// TwinCAT 3 PLC project PLC
// ProgramVersion: 3.1.4024.0
// libraries:
//   EfficientIO Communicator, * (EfficientIO)
//   Lynus Energy Basic, * (Lynus AG)
//   Lynus Persistent Data V1, * (Lynus AG)
//   Lynus Standards, * (Lynus AG)
//   Tc2_Standard, * (Beckhoff Automation GmbH)
//   Tc2_System, * (Beckhoff Automation GmbH)
//   Tc3_IPCDiag, * (Beckhoff Automation GmbH)
//   Tc3_Module, * (Beckhoff Automation GmbH)
// project tree:
//   ENUMs/ E_State.TcDUT (not stored)
//   / FastTask.TcTTO, MiddleTask.TcTTO, SlowTask.TcTTO (not stored)
//   POUs/ prgComEffIO.TcPOU, prgEM.TcPOU, prgOutputs.TcPOU, prgRWEffIO.TcPOU (not stored), prgVarEffIO.TcPOU (not stored), prg_ReadDeviceName.TcPOU (not stored)
// real-time tasks:
//   TASK PlcTask: cycle T#10ms, priority 20, ADS port 350
//   TASK FastTask: cycle T#5ms, priority 19, ADS port 351
//   TASK MiddleTask: cycle T#10ms, priority 21, ADS port 352
//   TASK SlowTask: cycle T#20ms, priority 23, ADS port 353
// I/O:
//   DEVICE Gerät 2 (CX-BK)
//     Box 1 (CX-BK)
// variable links:
//   PLC/PLC Instance <-> Device 2 (CX-BK)/Box 1 (CX-BK)
//     MiddleTask Inputs/prgEM.fbEM1.fbKL3403.byStateCH1 <-> Term 2 (KL3403)/Channel 1/Status
//     MiddleTask Inputs/prgEM.fbEM1.fbKL3403.byStateCH2 <-> Term 2 (KL3403)/Channel 2/Status
//     MiddleTask Inputs/prgEM.fbEM1.fbKL3403.byStateCH3 <-> Term 2 (KL3403)/Channel 3/Status
//     MiddleTask Inputs/prgEM.fbEM10.fbKL3403.byStateCH1 <-> Term 11 (KL3403)/Channel 1/Status
//     MiddleTask Inputs/prgEM.fbEM10.fbKL3403.byStateCH2 <-> Term 11 (KL3403)/Channel 2/Status
//     MiddleTask Inputs/prgEM.fbEM10.fbKL3403.byStateCH3 <-> Term 11 (KL3403)/Channel 3/Status
//     MiddleTask Inputs/prgEM.fbEM11.fbKL3403.byStateCH1 <-> Term 12 (KL3403)/Channel 1/Status
//     MiddleTask Inputs/prgEM.fbEM11.fbKL3403.byStateCH2 <-> Term 12 (KL3403)/Channel 2/Status
//     MiddleTask Inputs/prgEM.fbEM11.fbKL3403.byStateCH3 <-> Term 12 (KL3403)/Channel 3/Status
//     MiddleTask Inputs/prgEM.fbEM12.fbKL3403.byStateCH1 <-> Term 13 (KL3403)/Channel 1/Status
//     MiddleTask Inputs/prgEM.fbEM12.fbKL3403.byStateCH2 <-> Term 13 (KL3403)/Channel 2/Status
//     MiddleTask Inputs/prgEM.fbEM12.fbKL3403.byStateCH3 <-> Term 13 (KL3403)/Channel 3/Status
//     MiddleTask Inputs/prgEM.fbEM2.fbKL3403.byStateCH1 <-> Term 3 (KL3403)/Channel 1/Status
//     MiddleTask Inputs/prgEM.fbEM2.fbKL3403.byStateCH2 <-> Term 3 (KL3403)/Channel 2/Status
//     MiddleTask Inputs/prgEM.fbEM2.fbKL3403.byStateCH3 <-> Term 3 (KL3403)/Channel 3/Status
//     MiddleTask Inputs/prgEM.fbEM3.fbKL3403.byStateCH1 <-> Term 4 (KL3403)/Channel 1/Status
//     MiddleTask Inputs/prgEM.fbEM3.fbKL3403.byStateCH2 <-> Term 4 (KL3403)/Channel 2/Status
//     MiddleTask Inputs/prgEM.fbEM3.fbKL3403.byStateCH3 <-> Term 4 (KL3403)/Channel 3/Status
//     MiddleTask Inputs/prgEM.fbEM4.fbKL3403.byStateCH1 <-> Term 5 (KL3403)/Channel 1/Status
//     MiddleTask Inputs/prgEM.fbEM4.fbKL3403.byStateCH2 <-> Term 5 (KL3403)/Channel 2/Status
//     MiddleTask Inputs/prgEM.fbEM4.fbKL3403.byStateCH3 <-> Term 5 (KL3403)/Channel 3/Status
//     MiddleTask Inputs/prgEM.fbEM5.fbKL3403.byStateCH1 <-> Term 6 (KL3403)/Channel 1/Status
//     MiddleTask Inputs/prgEM.fbEM5.fbKL3403.byStateCH2 <-> Term 6 (KL3403)/Channel 2/Status
//     MiddleTask Inputs/prgEM.fbEM5.fbKL3403.byStateCH3 <-> Term 6 (KL3403)/Channel 3/Status
//     MiddleTask Inputs/prgEM.fbEM6.fbKL3403.byStateCH1 <-> Term 7 (KL3403)/Channel 1/Status
//     MiddleTask Inputs/prgEM.fbEM6.fbKL3403.byStateCH2 <-> Term 7 (KL3403)/Channel 2/Status
//     MiddleTask Inputs/prgEM.fbEM6.fbKL3403.byStateCH3 <-> Term 7 (KL3403)/Channel 3/Status
//     MiddleTask Inputs/prgEM.fbEM7.fbKL3403.byStateCH1 <-> Term 8 (KL3403)/Channel 1/Status
//     MiddleTask Inputs/prgEM.fbEM7.fbKL3403.byStateCH2 <-> Term 8 (KL3403)/Channel 2/Status
//     MiddleTask Inputs/prgEM.fbEM7.fbKL3403.byStateCH3 <-> Term 8 (KL3403)/Channel 3/Status
//     MiddleTask Inputs/prgEM.fbEM8.fbKL3403.byStateCH1 <-> Term 9 (KL3403)/Channel 1/Status
//     MiddleTask Inputs/prgEM.fbEM8.fbKL3403.byStateCH2 <-> Term 9 (KL3403)/Channel 2/Status
//     MiddleTask Inputs/prgEM.fbEM8.fbKL3403.byStateCH3 <-> Term 9 (KL3403)/Channel 3/Status
//     MiddleTask Inputs/prgEM.fbEM9.fbKL3403.byStateCH1 <-> Term 10 (KL3403)/Channel 1/Status
//     MiddleTask Inputs/prgEM.fbEM9.fbKL3403.byStateCH2 <-> Term 10 (KL3403)/Channel 2/Status
//     MiddleTask Inputs/prgEM.fbEM9.fbKL3403.byStateCH3 <-> Term 10 (KL3403)/Channel 3/Status
//     MiddleTask Inputs/prgEM.fbEM1.fbKL3403.iDataInCH1 <-> Term 2 (KL3403)/Channel 1/Daten Ein
//     MiddleTask Inputs/prgEM.fbEM1.fbKL3403.iDataInCH2 <-> Term 2 (KL3403)/Channel 2/Daten Ein
//     MiddleTask Inputs/prgEM.fbEM1.fbKL3403.iDataInCH3 <-> Term 2 (KL3403)/Channel 3/Daten Ein
//     MiddleTask Inputs/prgEM.fbEM10.fbKL3403.iDataInCH1 <-> Term 11 (KL3403)/Channel 1/Daten Ein
//     MiddleTask Inputs/prgEM.fbEM10.fbKL3403.iDataInCH2 <-> Term 11 (KL3403)/Channel 2/Daten Ein
//     MiddleTask Inputs/prgEM.fbEM10.fbKL3403.iDataInCH3 <-> Term 11 (KL3403)/Channel 3/Daten Ein
//     MiddleTask Inputs/prgEM.fbEM11.fbKL3403.iDataInCH1 <-> Term 12 (KL3403)/Channel 1/Daten Ein
//     MiddleTask Inputs/prgEM.fbEM11.fbKL3403.iDataInCH2 <-> Term 12 (KL3403)/Channel 2/Daten Ein
//     MiddleTask Inputs/prgEM.fbEM11.fbKL3403.iDataInCH3 <-> Term 12 (KL3403)/Channel 3/Daten Ein
//     MiddleTask Inputs/prgEM.fbEM12.fbKL3403.iDataInCH1 <-> Term 13 (KL3403)/Channel 1/Daten Ein
//     MiddleTask Inputs/prgEM.fbEM12.fbKL3403.iDataInCH2 <-> Term 13 (KL3403)/Channel 2/Daten Ein
//     MiddleTask Inputs/prgEM.fbEM12.fbKL3403.iDataInCH3 <-> Term 13 (KL3403)/Channel 3/Daten Ein
//     MiddleTask Inputs/prgEM.fbEM2.fbKL3403.iDataInCH1 <-> Term 3 (KL3403)/Channel 1/Daten Ein
//     MiddleTask Inputs/prgEM.fbEM2.fbKL3403.iDataInCH2 <-> Term 3 (KL3403)/Channel 2/Daten Ein
//     MiddleTask Inputs/prgEM.fbEM2.fbKL3403.iDataInCH3 <-> Term 3 (KL3403)/Channel 3/Daten Ein
//     MiddleTask Inputs/prgEM.fbEM3.fbKL3403.iDataInCH1 <-> Term 4 (KL3403)/Channel 1/Daten Ein
//     MiddleTask Inputs/prgEM.fbEM3.fbKL3403.iDataInCH2 <-> Term 4 (KL3403)/Channel 2/Daten Ein
//     MiddleTask Inputs/prgEM.fbEM3.fbKL3403.iDataInCH3 <-> Term 4 (KL3403)/Channel 3/Daten Ein
//     MiddleTask Inputs/prgEM.fbEM4.fbKL3403.iDataInCH1 <-> Term 5 (KL3403)/Channel 1/Daten Ein
//     MiddleTask Inputs/prgEM.fbEM4.fbKL3403.iDataInCH2 <-> Term 5 (KL3403)/Channel 2/Daten Ein
//     MiddleTask Inputs/prgEM.fbEM4.fbKL3403.iDataInCH3 <-> Term 5 (KL3403)/Channel 3/Daten Ein
//     MiddleTask Inputs/prgEM.fbEM5.fbKL3403.iDataInCH1 <-> Term 6 (KL3403)/Channel 1/Daten Ein
//     MiddleTask Inputs/prgEM.fbEM5.fbKL3403.iDataInCH2 <-> Term 6 (KL3403)/Channel 2/Daten Ein
//     MiddleTask Inputs/prgEM.fbEM5.fbKL3403.iDataInCH3 <-> Term 6 (KL3403)/Channel 3/Daten Ein
//     MiddleTask Inputs/prgEM.fbEM6.fbKL3403.iDataInCH1 <-> Term 7 (KL3403)/Channel 1/Daten Ein
//     MiddleTask Inputs/prgEM.fbEM6.fbKL3403.iDataInCH2 <-> Term 7 (KL3403)/Channel 2/Daten Ein
//     MiddleTask Inputs/prgEM.fbEM6.fbKL3403.iDataInCH3 <-> Term 7 (KL3403)/Channel 3/Daten Ein
//     MiddleTask Inputs/prgEM.fbEM7.fbKL3403.iDataInCH1 <-> Term 8 (KL3403)/Channel 1/Daten Ein
//     MiddleTask Inputs/prgEM.fbEM7.fbKL3403.iDataInCH2 <-> Term 8 (KL3403)/Channel 2/Daten Ein
//     MiddleTask Inputs/prgEM.fbEM7.fbKL3403.iDataInCH3 <-> Term 8 (KL3403)/Channel 3/Daten Ein
//     MiddleTask Inputs/prgEM.fbEM8.fbKL3403.iDataInCH1 <-> Term 9 (KL3403)/Channel 1/Daten Ein
//     MiddleTask Inputs/prgEM.fbEM8.fbKL3403.iDataInCH2 <-> Term 9 (KL3403)/Channel 2/Daten Ein
//     MiddleTask Inputs/prgEM.fbEM8.fbKL3403.iDataInCH3 <-> Term 9 (KL3403)/Channel 3/Daten Ein
//     MiddleTask Inputs/prgEM.fbEM9.fbKL3403.iDataInCH1 <-> Term 10 (KL3403)/Channel 1/Daten Ein
//     MiddleTask Inputs/prgEM.fbEM9.fbKL3403.iDataInCH2 <-> Term 10 (KL3403)/Channel 2/Daten Ein
//     MiddleTask Inputs/prgEM.fbEM9.fbKL3403.iDataInCH3 <-> Term 10 (KL3403)/Channel 3/Daten Ein
//     MiddleTask Inputs/prgEM.fbKBusState.uiKBusState_OUT <-> Inputs/State
//     MiddleTask Outputs/prgEM.fbEM1.fbKL3403.byCntrCH1 <-> Term 2 (KL3403)/Channel 1/Kontrolle
//     MiddleTask Outputs/prgEM.fbEM1.fbKL3403.byCntrCH2 <-> Term 2 (KL3403)/Channel 2/Kontrolle
//     MiddleTask Outputs/prgEM.fbEM1.fbKL3403.byCntrCH3 <-> Term 2 (KL3403)/Channel 3/Kontrolle
//     MiddleTask Outputs/prgEM.fbEM10.fbKL3403.byCntrCH1 <-> Term 11 (KL3403)/Channel 1/Kontrolle
//     MiddleTask Outputs/prgEM.fbEM10.fbKL3403.byCntrCH2 <-> Term 11 (KL3403)/Channel 2/Kontrolle
//     MiddleTask Outputs/prgEM.fbEM10.fbKL3403.byCntrCH3 <-> Term 11 (KL3403)/Channel 3/Kontrolle
//     MiddleTask Outputs/prgEM.fbEM11.fbKL3403.byCntrCH1 <-> Term 12 (KL3403)/Channel 1/Kontrolle
//     MiddleTask Outputs/prgEM.fbEM11.fbKL3403.byCntrCH2 <-> Term 12 (KL3403)/Channel 2/Kontrolle
//     MiddleTask Outputs/prgEM.fbEM11.fbKL3403.byCntrCH3 <-> Term 12 (KL3403)/Channel 3/Kontrolle
//     MiddleTask Outputs/prgEM.fbEM12.fbKL3403.byCntrCH1 <-> Term 13 (KL3403)/Channel 1/Kontrolle
//     MiddleTask Outputs/prgEM.fbEM12.fbKL3403.byCntrCH2 <-> Term 13 (KL3403)/Channel 2/Kontrolle
//     MiddleTask Outputs/prgEM.fbEM12.fbKL3403.byCntrCH3 <-> Term 13 (KL3403)/Channel 3/Kontrolle
//     MiddleTask Outputs/prgEM.fbEM2.fbKL3403.byCntrCH1 <-> Term 3 (KL3403)/Channel 1/Kontrolle
//     MiddleTask Outputs/prgEM.fbEM2.fbKL3403.byCntrCH2 <-> Term 3 (KL3403)/Channel 2/Kontrolle
//     MiddleTask Outputs/prgEM.fbEM2.fbKL3403.byCntrCH3 <-> Term 3 (KL3403)/Channel 3/Kontrolle
//     MiddleTask Outputs/prgEM.fbEM3.fbKL3403.byCntrCH1 <-> Term 4 (KL3403)/Channel 1/Kontrolle
//     MiddleTask Outputs/prgEM.fbEM3.fbKL3403.byCntrCH2 <-> Term 4 (KL3403)/Channel 2/Kontrolle
//     MiddleTask Outputs/prgEM.fbEM3.fbKL3403.byCntrCH3 <-> Term 4 (KL3403)/Channel 3/Kontrolle
//     MiddleTask Outputs/prgEM.fbEM4.fbKL3403.byCntrCH1 <-> Term 5 (KL3403)/Channel 1/Kontrolle
//     MiddleTask Outputs/prgEM.fbEM4.fbKL3403.byCntrCH2 <-> Term 5 (KL3403)/Channel 2/Kontrolle
//     MiddleTask Outputs/prgEM.fbEM4.fbKL3403.byCntrCH3 <-> Term 5 (KL3403)/Channel 3/Kontrolle
//     MiddleTask Outputs/prgEM.fbEM5.fbKL3403.byCntrCH1 <-> Term 6 (KL3403)/Channel 1/Kontrolle
//     MiddleTask Outputs/prgEM.fbEM5.fbKL3403.byCntrCH2 <-> Term 6 (KL3403)/Channel 2/Kontrolle
//     MiddleTask Outputs/prgEM.fbEM5.fbKL3403.byCntrCH3 <-> Term 6 (KL3403)/Channel 3/Kontrolle
//     MiddleTask Outputs/prgEM.fbEM6.fbKL3403.byCntrCH1 <-> Term 7 (KL3403)/Channel 1/Kontrolle
//     MiddleTask Outputs/prgEM.fbEM6.fbKL3403.byCntrCH2 <-> Term 7 (KL3403)/Channel 2/Kontrolle
//     MiddleTask Outputs/prgEM.fbEM6.fbKL3403.byCntrCH3 <-> Term 7 (KL3403)/Channel 3/Kontrolle
//     MiddleTask Outputs/prgEM.fbEM7.fbKL3403.byCntrCH1 <-> Term 8 (KL3403)/Channel 1/Kontrolle
//     MiddleTask Outputs/prgEM.fbEM7.fbKL3403.byCntrCH2 <-> Term 8 (KL3403)/Channel 2/Kontrolle
//     MiddleTask Outputs/prgEM.fbEM7.fbKL3403.byCntrCH3 <-> Term 8 (KL3403)/Channel 3/Kontrolle
//     MiddleTask Outputs/prgEM.fbEM8.fbKL3403.byCntrCH1 <-> Term 9 (KL3403)/Channel 1/Kontrolle
//     MiddleTask Outputs/prgEM.fbEM8.fbKL3403.byCntrCH2 <-> Term 9 (KL3403)/Channel 2/Kontrolle
//     MiddleTask Outputs/prgEM.fbEM8.fbKL3403.byCntrCH3 <-> Term 9 (KL3403)/Channel 3/Kontrolle
//     MiddleTask Outputs/prgEM.fbEM9.fbKL3403.byCntrCH1 <-> Term 10 (KL3403)/Channel 1/Kontrolle
//     MiddleTask Outputs/prgEM.fbEM9.fbKL3403.byCntrCH2 <-> Term 10 (KL3403)/Channel 2/Kontrolle
//     MiddleTask Outputs/prgEM.fbEM9.fbKL3403.byCntrCH3 <-> Term 10 (KL3403)/Channel 3/Kontrolle
//     MiddleTask Outputs/prgOutputs.mOut_1_1 <-> Term 14 (KL2012)/Channel 1/Ausgang
//     MiddleTask Outputs/prgOutputs.mOut_1_2 <-> Term 14 (KL2012)/Channel 2/Ausgang
//     MiddleTask Outputs/prgOutputs.mOut_2_1 <-> Term 15 (KL2012)/Channel 1/Ausgang
//     MiddleTask Outputs/prgOutputs.mOut_2_2 <-> Term 15 (KL2012)/Channel 2/Ausgang
//     MiddleTask Outputs/prgOutputs.mOut_3_1 <-> Term 16 (KL2012)/Channel 1/Ausgang
//     MiddleTask Outputs/prgOutputs.mOut_3_2 <-> Term 16 (KL2012)/Channel 2/Ausgang
//     MiddleTask Outputs/prgOutputs.mOut_4_1 <-> Term 17 (KL2012)/Channel 1/Ausgang
//     MiddleTask Outputs/prgOutputs.mOut_4_2 <-> Term 17 (KL2012)/Channel 2/Ausgang

CONFIGURATION PLC
    RESOURCE PLC ON TwinCAT3
        TASK FastTask(INTERVAL := T#5ms, PRIORITY := 19);
        TASK MiddleTask(INTERVAL := T#10ms, PRIORITY := 21);
        PROGRAM prgRWEffIO WITH FastTask : prgRWEffIO;
        PROGRAM prgVarEffIO WITH FastTask : prgVarEffIO;
        PROGRAM prgEM WITH MiddleTask : prgEM;
        PROGRAM prgOutputs WITH MiddleTask : prgOutputs;
    END_RESOURCE
END_CONFIGURATION

// ---- POUs/prgEM.TcPOU
PROGRAM prgEM
VAR
	fbKBusState		: FB_K_Bus_State;
	fbEM1			: FB_EM_Beckhoff_KL3403;
	fbEM1Counter	: FB_EnergyCounter;
	fbEM2			: FB_EM_Beckhoff_KL3403;
	fbEM2Counter	: FB_EnergyCounter;
	fbEM3			: FB_EM_Beckhoff_KL3403;
	fbEM3Counter	: FB_EnergyCounter;
	fbEM4			: FB_EM_Beckhoff_KL3403;
	fbEM4Counter	: FB_EnergyCounter;
	fbEM5			: FB_EM_Beckhoff_KL3403;
	fbEM5Counter	: FB_EnergyCounter;
	fbEM6			: FB_EM_Beckhoff_KL3403;
	fbEM6Counter	: FB_EnergyCounter;
	fbEM7			: FB_EM_Beckhoff_KL3403;
	fbEM7Counter	: FB_EnergyCounter;
	fbEM8			: FB_EM_Beckhoff_KL3403;
	fbEM8Counter	: FB_EnergyCounter;
	fbEM9			: FB_EM_Beckhoff_KL3403;
	fbEM9Counter	: FB_EnergyCounter;
	fbEM10			: FB_EM_Beckhoff_KL3403;
	fbEM10Counter	: FB_EnergyCounter;
	fbEM11			: FB_EM_Beckhoff_KL3403;
	fbEM11Counter	: FB_EnergyCounter;
	fbEM12			: FB_EM_Beckhoff_KL3403;
	fbEM12Counter	: FB_EnergyCounter;
	
	lrPowerEM1		: LREAL;						//{#lynus.ag#()}
	lrPowerEM2		: LREAL;						//{#lynus.ag#()}
	lrPowerEM3		: LREAL;						//{#lynus.ag#()}
	lrPowerEM4		: LREAL;						//{#lynus.ag#()}
	lrPowerEM5		: LREAL;						//{#lynus.ag#()}
	lrPowerEM6		: LREAL;						//{#lynus.ag#()}
	lrPowerEM7		: LREAL;						//{#lynus.ag#()}
	lrPowerEM8		: LREAL;						//{#lynus.ag#()}
	lrPowerEM9		: LREAL;						//{#lynus.ag#()}
	lrPowerEM10		: LREAL;						//{#lynus.ag#()}
	lrPowerEM11		: LREAL;						//{#lynus.ag#()}
	lrPowerEM12		: LREAL;						//{#lynus.ag#()}
	lr_InputVoltage_L1N		: LREAL;						//{#lynus.ag#()}
	lr_InputVoltage_L2N		: LREAL;						//{#lynus.ag#()}
	lr_InputVoltage_L3N		: LREAL;						//{#lynus.ag#()}
	lr_InputVoltage_L1L2	: LREAL;						//{#lynus.ag#()}
	lr_InputVoltage_L2L3	: LREAL;						//{#lynus.ag#()}
	lr_InputVoltage_L3L1	: LREAL;						//{#lynus.ag#()}
	lr_FrequencyEM1			: LREAL;						//{#lynus.ag#()}
	lr_CurrentL1EM1			: LREAL;						//{#lynus.ag#()}
	lr_CurrentL2EM1			: LREAL;						//{#lynus.ag#()}
	lr_CurrentL3EM1			: LREAL;						//{#lynus.ag#()}
END_VAR
VAR_INPUT
	uiCurrentTransformerRatio_EM1	:UINT:=400;			// unklar ob korrekt
	uiCurrentTransformerRatio_EM2	:UINT:=400;			// unklar ob korrekt
	uiCurrentTransformerRatio_EM3	:UINT:=250;
	uiCurrentTransformerRatio_EM4	:UINT:=64;
	uiCurrentTransformerRatio_EM5	:UINT:=64;
	uiCurrentTransformerRatio_EM6	:UINT:=35;
	uiCurrentTransformerRatio_EM7	:UINT:=35;
	uiCurrentTransformerRatio_EM8	:UINT:=35;
	uiCurrentTransformerRatio_EM9	:UINT:=35;
	uiCurrentTransformerRatio_EM10	:UINT:=35;
	uiCurrentTransformerRatio_EM11	:UINT:=35;
	uiCurrentTransformerRatio_EM12	:UINT:=35;

END_VAR
VAR PERSISTENT
	lrCounterEM1	: LREAL;						//{#lynus.ag#()}
	lrCounterEM2	: LREAL;						//{#lynus.ag#()}
	lrCounterEM3	: LREAL;						//{#lynus.ag#()}
	lrCounterEM4	: LREAL;						//{#lynus.ag#()}
	lrCounterEM5	: LREAL;						//{#lynus.ag#()}
	lrCounterEM6	: LREAL;						//{#lynus.ag#()}
	lrCounterEM7	: LREAL;						//{#lynus.ag#()}
	lrCounterEM8	: LREAL;						//{#lynus.ag#()}
	lrCounterEM9	: LREAL;						//{#lynus.ag#()}
	lrCounterEM10	: LREAL;						//{#lynus.ag#()}
	lrCounterEM11	: LREAL;						//{#lynus.ag#()}
	lrCounterEM12	: LREAL;						//{#lynus.ag#()}
END_VAR

fbKBusState(	uiKBusState_OUT=> , 
				b_Kbus_notOk=> , 
				word_ErrorCount=> );


fbEM1(
	bEnable:= TRUE, 
	bChannel1Invers:= FALSE,
	bChannel2Invers:= FALSE,
	bChannel3Invers:= FALSE,
	uiCurrentTransformerRatioL1:= uiCurrentTransformerRatio_EM1, 
	uiCurrentTransformerRatioL2:= uiCurrentTransformerRatio_EM1, 
	uiCurrentTransformerRatioL3:= uiCurrentTransformerRatio_EM1, 
	uiKBusState_IN:= fbKBusState.uiKBusState_OUT, 
	stDataEMPower=> , 
	stDataEMCounter=> , 
	stDataEMPowerRealTime=> , 
	stDataEMCounterRealTime=> , 
	diNrOfEM_OUT=> );

lrPowerEM1 := fbEM1.stDataEMPower.lrPowerTotal;	
lr_InputVoltage_L1N := fbEM1.stDataEMPower.lrVoltageL1N;
lr_InputVoltage_L2N := fbEM1.stDataEMPower.lrVoltageL2N;
lr_InputVoltage_L3N := fbEM1.stDataEMPower.lrVoltageL3N;
lr_InputVoltage_L1L2 := fbEM1.stDataEMPower.lrVoltageL1L2;
lr_InputVoltage_L2L3 := fbEM1.stDataEMPower.lrVoltageL2L3;
lr_InputVoltage_L3L1 := fbEM1.stDataEMPower.lrVoltageL3L1;
lr_FrequencyEM1		:= fbEM1.stDataEMPower.lrFrequency;
lr_CurrentL1EM1		:= fbEM1.stDataEMPower.lrCurrentL1;
lr_CurrentL2EM1		:= fbEM1.stDataEMPower.lrCurrentL2;
lr_CurrentL3EM1		:= fbEM1.stDataEMPower.lrCurrentL3;

fbEM1Counter(
	byActiveTariff:= 1, 
	lrPowerInput:= lrPowerEM1, 
	lrTotalCounterEnergy_Consumption=> , 
	lrTotalCounterEnergy_Production=> , 
	lrCounterEnergyT1_Consumption=> , 
	lrCounterEnergyT2_Consumption=> , 
	lrCounterEnergyT1_Production=> , 
	lrCounterEnergyT2_Production=> );
	
IF fbEM1Counter.lrTotalCounterEnergy_Consumption > lrCounterEM1 THEN  	
	lrCounterEM1 := fbEM1Counter.lrTotalCounterEnergy_Consumption;
END_IF


fbEM2(
	bEnable:= TRUE, 
	bChannel1Invers:= FALSE,
	bChannel2Invers:= FALSE,
	bChannel3Invers:= FALSE,
	uiCurrentTransformerRatioL1:= uiCurrentTransformerRatio_EM2, 
	uiCurrentTransformerRatioL2:= uiCurrentTransformerRatio_EM2, 
	uiCurrentTransformerRatioL3:= uiCurrentTransformerRatio_EM2, 
	uiKBusState_IN:= fbKBusState.uiKBusState_OUT, 
	stDataEMPower=> , 
	stDataEMCounter=> , 
	stDataEMPowerRealTime=> , 
	stDataEMCounterRealTime=> , 
	diNrOfEM_OUT=> );

lrPowerEM2 := fbEM2.stDataEMPower.lrPowerTotal;	

fbEM2Counter(
	byActiveTariff:= 1, 
	lrPowerInput:= lrPowerEM2, 
	lrTotalCounterEnergy_Consumption=> , 
	lrTotalCounterEnergy_Production=> , 
	lrCounterEnergyT1_Consumption=> , 
	lrCounterEnergyT2_Consumption=> , 
	lrCounterEnergyT1_Production=> , 
	lrCounterEnergyT2_Production=> );
	
IF fbEM2Counter.lrTotalCounterEnergy_Consumption > lrCounterEM2 THEN  	
	lrCounterEM2 := fbEM2Counter.lrTotalCounterEnergy_Consumption;
END_IF


fbEM3(
	bEnable:= TRUE, 
	bChannel1Invers:= FALSE,
	bChannel2Invers:= FALSE,
	bChannel3Invers:= FALSE,
	uiCurrentTransformerRatioL1:= uiCurrentTransformerRatio_EM3, 
	uiCurrentTransformerRatioL2:= uiCurrentTransformerRatio_EM3, 
	uiCurrentTransformerRatioL3:= uiCurrentTransformerRatio_EM3, 
	uiKBusState_IN:= fbKBusState.uiKBusState_OUT, 
	stDataEMPower=> , 
	stDataEMCounter=> , 
	stDataEMPowerRealTime=> , 
	stDataEMCounterRealTime=> , 
	diNrOfEM_OUT=> );

lrPowerEM3 := fbEM3.stDataEMPower.lrPowerTotal;	

fbEM3Counter(
	byActiveTariff:= 1, 
	lrPowerInput:= lrPowerEM3, 
	lrTotalCounterEnergy_Consumption=> , 
	lrTotalCounterEnergy_Production=> , 
	lrCounterEnergyT1_Consumption=> , 
	lrCounterEnergyT2_Consumption=> , 
	lrCounterEnergyT1_Production=> , 
	lrCounterEnergyT2_Production=> );
	
IF fbEM3Counter.lrTotalCounterEnergy_Consumption > lrCounterEM3 THEN  	
	lrCounterEM3 := fbEM3Counter.lrTotalCounterEnergy_Consumption;
END_IF

fbEM4(
	bEnable:= TRUE, 
	bChannel1Invers:= FALSE,
	bChannel2Invers:= FALSE,
	bChannel3Invers:= FALSE,
	uiCurrentTransformerRatioL1:= uiCurrentTransformerRatio_EM4, 
	uiCurrentTransformerRatioL2:= uiCurrentTransformerRatio_EM4, 
	uiCurrentTransformerRatioL3:= uiCurrentTransformerRatio_EM4, 
	uiKBusState_IN:= fbKBusState.uiKBusState_OUT, 
	stDataEMPower=> , 
	stDataEMCounter=> , 
	stDataEMPowerRealTime=> , 
	stDataEMCounterRealTime=> , 
	diNrOfEM_OUT=> );

lrPowerEM4 := fbEM4.stDataEMPower.lrPowerTotal;	

fbEM4Counter(
	byActiveTariff:= 1, 
	lrPowerInput:= lrPowerEM4, 
	lrTotalCounterEnergy_Consumption=> , 
	lrTotalCounterEnergy_Production=> , 
	lrCounterEnergyT1_Consumption=> , 
	lrCounterEnergyT2_Consumption=> , 
	lrCounterEnergyT1_Production=> , 
	lrCounterEnergyT2_Production=> );
	
IF fbEM4Counter.lrTotalCounterEnergy_Consumption > lrCounterEM4 THEN  	
	lrCounterEM4 := fbEM4Counter.lrTotalCounterEnergy_Consumption;
END_IF

fbEM5(
	bEnable:= TRUE, 
	bChannel1Invers:= FALSE,
	bChannel2Invers:= FALSE,
	bChannel3Invers:= FALSE,
	uiCurrentTransformerRatioL1:= uiCurrentTransformerRatio_EM5, 
	uiCurrentTransformerRatioL2:= uiCurrentTransformerRatio_EM5, 
	uiCurrentTransformerRatioL3:= uiCurrentTransformerRatio_EM5, 
	uiKBusState_IN:= fbKBusState.uiKBusState_OUT, 
	stDataEMPower=> , 
	stDataEMCounter=> , 
	stDataEMPowerRealTime=> , 
	stDataEMCounterRealTime=> , 
	diNrOfEM_OUT=> );

lrPowerEM5 := fbEM5.stDataEMPower.lrPowerTotal;	

fbEM5Counter(
	byActiveTariff:= 1, 
	lrPowerInput:= lrPowerEM5, 
	lrTotalCounterEnergy_Consumption=> , 
	lrTotalCounterEnergy_Production=> , 
	lrCounterEnergyT1_Consumption=> , 
	lrCounterEnergyT2_Consumption=> , 
	lrCounterEnergyT1_Production=> , 
	lrCounterEnergyT2_Production=> );
	
IF fbEM5Counter.lrTotalCounterEnergy_Consumption > lrCounterEM5 THEN  	
	lrCounterEM5 := fbEM5Counter.lrTotalCounterEnergy_Consumption;
END_IF

fbEM6(
	bEnable:= TRUE, 
	bChannel1Invers:= FALSE,
	bChannel2Invers:= FALSE,
	bChannel3Invers:= FALSE,
	uiCurrentTransformerRatioL1:= uiCurrentTransformerRatio_EM6, 
	uiCurrentTransformerRatioL2:= uiCurrentTransformerRatio_EM6, 
	uiCurrentTransformerRatioL3:= uiCurrentTransformerRatio_EM6, 
	uiKBusState_IN:= fbKBusState.uiKBusState_OUT, 
	stDataEMPower=> , 
	stDataEMCounter=> , 
	stDataEMPowerRealTime=> , 
	stDataEMCounterRealTime=> , 
	diNrOfEM_OUT=> );

lrPowerEM6 := fbEM6.stDataEMPower.lrPowerTotal;	

fbEM6Counter(
	byActiveTariff:= 1, 
	lrPowerInput:= lrPowerEM6, 
	lrTotalCounterEnergy_Consumption=> , 
	lrTotalCounterEnergy_Production=> , 
	lrCounterEnergyT1_Consumption=> , 
	lrCounterEnergyT2_Consumption=> , 
	lrCounterEnergyT1_Production=> , 
	lrCounterEnergyT2_Production=> );
	
IF fbEM6Counter.lrTotalCounterEnergy_Consumption > lrCounterEM6 THEN  	
	lrCounterEM6 := fbEM6Counter.lrTotalCounterEnergy_Consumption;
END_IF

fbEM7(
	bEnable:= TRUE, 
	bChannel1Invers:= FALSE,
	bChannel2Invers:= FALSE,
	bChannel3Invers:= FALSE,
	uiCurrentTransformerRatioL1:= uiCurrentTransformerRatio_EM7, 
	uiCurrentTransformerRatioL2:= uiCurrentTransformerRatio_EM7, 
	uiCurrentTransformerRatioL3:= uiCurrentTransformerRatio_EM7, 
	uiKBusState_IN:= fbKBusState.uiKBusState_OUT, 
	stDataEMPower=> , 
	stDataEMCounter=> , 
	stDataEMPowerRealTime=> , 
	stDataEMCounterRealTime=> , 
	diNrOfEM_OUT=> );

lrPowerEM7 := fbEM7.stDataEMPower.lrPowerTotal;	

fbEM7Counter(
	byActiveTariff:= 1, 
	lrPowerInput:= lrPowerEM7, 
	lrTotalCounterEnergy_Consumption=> , 
	lrTotalCounterEnergy_Production=> , 
	lrCounterEnergyT1_Consumption=> , 
	lrCounterEnergyT2_Consumption=> , 
	lrCounterEnergyT1_Production=> , 
	lrCounterEnergyT2_Production=> );
	
IF fbEM7Counter.lrTotalCounterEnergy_Consumption > lrCounterEM7 THEN  	
	lrCounterEM7 := fbEM7Counter.lrTotalCounterEnergy_Consumption;
END_IF

fbEM8(
	bEnable:= TRUE, 
	bChannel1Invers:= FALSE,
	bChannel2Invers:= FALSE,
	bChannel3Invers:= FALSE,
	uiCurrentTransformerRatioL1:= uiCurrentTransformerRatio_EM8, 
	uiCurrentTransformerRatioL2:= uiCurrentTransformerRatio_EM8, 
	uiCurrentTransformerRatioL3:= uiCurrentTransformerRatio_EM8, 
	uiKBusState_IN:= fbKBusState.uiKBusState_OUT, 
	stDataEMPower=> , 
	stDataEMCounter=> , 
	stDataEMPowerRealTime=> , 
	stDataEMCounterRealTime=> , 
	diNrOfEM_OUT=> );

lrPowerEM8 := fbEM8.stDataEMPower.lrPowerTotal;	

fbEM8Counter(
	byActiveTariff:= 1, 
	lrPowerInput:= lrPowerEM8, 
	lrTotalCounterEnergy_Consumption=> , 
	lrTotalCounterEnergy_Production=> , 
	lrCounterEnergyT1_Consumption=> , 
	lrCounterEnergyT2_Consumption=> , 
	lrCounterEnergyT1_Production=> , 
	lrCounterEnergyT2_Production=> );
	
IF fbEM8Counter.lrTotalCounterEnergy_Consumption > lrCounterEM8 THEN  	
	lrCounterEM8 := fbEM8Counter.lrTotalCounterEnergy_Consumption;
END_IF

fbEM9(
	bEnable:= TRUE, 
	bChannel1Invers:= FALSE,
	bChannel2Invers:= FALSE,
	bChannel3Invers:= FALSE,
	uiCurrentTransformerRatioL1:= uiCurrentTransformerRatio_EM9, 
	uiCurrentTransformerRatioL2:= uiCurrentTransformerRatio_EM9, 
	uiCurrentTransformerRatioL3:= uiCurrentTransformerRatio_EM9, 
	uiKBusState_IN:= fbKBusState.uiKBusState_OUT, 
	stDataEMPower=> , 
	stDataEMCounter=> , 
	stDataEMPowerRealTime=> , 
	stDataEMCounterRealTime=> , 
	diNrOfEM_OUT=> );

lrPowerEM9 := fbEM9.stDataEMPower.lrPowerTotal;	

fbEM9Counter(
	byActiveTariff:= 1, 
	lrPowerInput:= lrPowerEM9, 
	lrTotalCounterEnergy_Consumption=> , 
	lrTotalCounterEnergy_Production=> , 
	lrCounterEnergyT1_Consumption=> , 
	lrCounterEnergyT2_Consumption=> , 
	lrCounterEnergyT1_Production=> , 
	lrCounterEnergyT2_Production=> );
	
IF fbEM9Counter.lrTotalCounterEnergy_Consumption > lrCounterEM9 THEN  	
	lrCounterEM9 := fbEM9Counter.lrTotalCounterEnergy_Consumption;
END_IF

fbEM10(
	bEnable:= TRUE, 
	bChannel1Invers:= FALSE,
	bChannel2Invers:= FALSE,
	bChannel3Invers:= FALSE,
	uiCurrentTransformerRatioL1:= uiCurrentTransformerRatio_EM10, 
	uiCurrentTransformerRatioL2:= uiCurrentTransformerRatio_EM10, 
	uiCurrentTransformerRatioL3:= uiCurrentTransformerRatio_EM10, 
	uiKBusState_IN:= fbKBusState.uiKBusState_OUT, 
	stDataEMPower=> , 
	stDataEMCounter=> , 
	stDataEMPowerRealTime=> , 
	stDataEMCounterRealTime=> , 
	diNrOfEM_OUT=> );

lrPowerEM10 := fbEM10.stDataEMPower.lrPowerTotal;	

fbEM10Counter(
	byActiveTariff:= 1, 
	lrPowerInput:= lrPowerEM10, 
	lrTotalCounterEnergy_Consumption=> , 
	lrTotalCounterEnergy_Production=> , 
	lrCounterEnergyT1_Consumption=> , 
	lrCounterEnergyT2_Consumption=> , 
	lrCounterEnergyT1_Production=> , 
	lrCounterEnergyT2_Production=> );
	
IF fbEM10Counter.lrTotalCounterEnergy_Consumption > lrCounterEM10 THEN  	
	lrCounterEM10 := fbEM10Counter.lrTotalCounterEnergy_Consumption;
END_IF

fbEM11(
	bEnable:= TRUE, 
	bChannel1Invers:= FALSE,
	bChannel2Invers:= FALSE,
	bChannel3Invers:= FALSE,
	uiCurrentTransformerRatioL1:= uiCurrentTransformerRatio_EM11, 
	uiCurrentTransformerRatioL2:= uiCurrentTransformerRatio_EM11, 
	uiCurrentTransformerRatioL3:= uiCurrentTransformerRatio_EM11, 
	uiKBusState_IN:= fbKBusState.uiKBusState_OUT, 
	stDataEMPower=> , 
	stDataEMCounter=> , 
	stDataEMPowerRealTime=> , 
	stDataEMCounterRealTime=> , 
	diNrOfEM_OUT=> );

lrPowerEM11 := fbEM11.stDataEMPower.lrPowerTotal;	

fbEM11Counter(
	byActiveTariff:= 1, 
	lrPowerInput:= lrPowerEM11, 
	lrTotalCounterEnergy_Consumption=> , 
	lrTotalCounterEnergy_Production=> , 
	lrCounterEnergyT1_Consumption=> , 
	lrCounterEnergyT2_Consumption=> , 
	lrCounterEnergyT1_Production=> , 
	lrCounterEnergyT2_Production=> );
	
IF fbEM11Counter.lrTotalCounterEnergy_Consumption > lrCounterEM11 THEN  	
	lrCounterEM11 := fbEM11Counter.lrTotalCounterEnergy_Consumption;
END_IF

fbEM12(
	bEnable:= TRUE, 
	bChannel1Invers:= FALSE,
	bChannel2Invers:= FALSE,
	bChannel3Invers:= FALSE,
	uiCurrentTransformerRatioL1:= uiCurrentTransformerRatio_EM12, 
	uiCurrentTransformerRatioL2:= uiCurrentTransformerRatio_EM12, 
	uiCurrentTransformerRatioL3:= uiCurrentTransformerRatio_EM12, 
	uiKBusState_IN:= fbKBusState.uiKBusState_OUT, 
	stDataEMPower=> , 
	stDataEMCounter=> , 
	stDataEMPowerRealTime=> , 
	stDataEMCounterRealTime=> , 
	diNrOfEM_OUT=> );

lrPowerEM12 := fbEM12.stDataEMPower.lrPowerTotal;	

fbEM12Counter(
	byActiveTariff:= 1, 
	lrPowerInput:= lrPowerEM12, 
	lrTotalCounterEnergy_Consumption=> , 
	lrTotalCounterEnergy_Production=> , 
	lrCounterEnergyT1_Consumption=> , 
	lrCounterEnergyT2_Consumption=> , 
	lrCounterEnergyT1_Production=> , 
	lrCounterEnergyT2_Production=> );
	
IF fbEM12Counter.lrTotalCounterEnergy_Consumption > lrCounterEM12 THEN  	
	lrCounterEM12 := fbEM12Counter.lrTotalCounterEnergy_Consumption;
END_IF

END_PROGRAM

// ---- POUs/prgOutputs.TcPOU
PROGRAM prgOutputs
VAR
	mOut_1_1		AT%Q*: BOOL;								//{#lynus.ag#()}
	mOut_1_2		AT%Q*: BOOL;								//{#lynus.ag#()}
	mOut_2_1		AT%Q*: BOOL;								//{#lynus.ag#()}
	mOut_2_2		AT%Q*: BOOL;								//{#lynus.ag#()}
	mOut_3_1		AT%Q*: BOOL;								//{#lynus.ag#()}
	mOut_3_2		AT%Q*: BOOL;								//{#lynus.ag#()}
	mOut_4_1		AT%Q*: BOOL;								//{#lynus.ag#()}
	mOut_4_2		AT%Q*: BOOL;								//{#lynus.ag#()}
	mOut_Command_1_1		:BOOL;								//{#lynus.ag#()}
	mOut_Command_1_2		:BOOL;								//{#lynus.ag#()}
	mOut_Command_2_1		:BOOL;								//{#lynus.ag#()}
	mOut_Command_2_2		:BOOL;								//{#lynus.ag#()}
	mOut_Command_3_1		:BOOL;								//{#lynus.ag#()}
	mOut_Command_3_2		:BOOL;								//{#lynus.ag#()}
	mOut_Command_4_1		:BOOL;								//{#lynus.ag#()}
	mOut_Command_4_2		:BOOL;								//{#lynus.ag#()}
END_VAR

mOut_1_1		:= 	mOut_Command_1_1;
mOut_1_2		:= 	mOut_Command_1_2;
mOut_2_1		:= 	mOut_Command_2_1;
mOut_2_2		:= 	mOut_Command_2_2;
mOut_3_1		:= 	mOut_Command_3_1;
mOut_3_2		:= 	mOut_Command_3_2;
mOut_4_1		:= 	mOut_Command_4_1;
mOut_4_2		:= 	mOut_Command_4_2;

END_PROGRAM

// ---- POUs/prgComEffIO.TcPOU
PROGRAM prgComEffIO
VAR
	fbCom		: FB_MqttCommunicator_V2;
	int_PowerLinkNumber: INT;
END_VAR

fbCom(
	bConnect:= TRUE, 
	strAuthkey := 'EIO08031879806',
	sUserName:= , 			// see below
	sUserPassword:= , 		// see below
	eSavePositionCertificate:= eSavePositionOnPLC.ePostionHardDisk, 
	bConnected=> , 
	bError=> , 
	hrErrorCode=> , 
	eConnectionState=> , 
	eErrorMessage_Out=> );



prg_ReadDeviceName();
IF prg_ReadDeviceName.sDeviceName = '' THEN
	prg_ReadDeviceName.bStart := TRUE;
END_IF

// select user / pass according device name:
 IF prg_ReadDeviceName.sDeviceName = 'EIOSP000002' THEN   // powerlink #1
	fbCom.sUserName:= 'bcb65b49-8b4d-4022-904c-9936d016ff1c'; 
	fbCom.sUserPassword:= 'd3bebec0-d67d-45ef-bae3-ebeb4a96c1a9';
	prgEM.uiCurrentTransformerRatio_EM1	:= 300;
	prgEM.uiCurrentTransformerRatio_EM2	:= 32;
	prgEM.uiCurrentTransformerRatio_EM3	:= 32;
	prgEM.uiCurrentTransformerRatio_EM4	:= 32;
	prgEM.uiCurrentTransformerRatio_EM5	:= 32;
	prgEM.uiCurrentTransformerRatio_EM6	:= 32;
	prgEM.uiCurrentTransformerRatio_EM7	:= 32;
	

END_IF

END_PROGRAM
